PROGRAM MAIN
VAR	
	ipImageMerge		:	ITcVnImage;
	ipImageRed			:	ITcVnImage;
	ipImageBlue			:	ITcVnImage;
	ipImageMergeDisp	:	ITcVnDisplayableImage;
	regionImageDisp	:	ITcVnDisplayableImage;
	
	aBlack				:	TcVnVector4_LREAL := [0, 0, 0];
	aRed				:	TcVnVector4_LREAL := [255, 0, 0];
	aBlue				:	TcVnVector4_LREAL := [0, 0, 255];
	
	aPositionRed		:	TcVnPoint := [20, 20];
	aPositionBlue		:	TcVnPoint := [480, 480];
	bCopyBlue			:	BOOL := FALSE;
	hr: DINT;
END_VAR

//	Disclaimer
  	
//	THIS publication contains statements about the suitability OF our products FOR certain 
//	areas OF application. These statements are based on typical features OF our products. 
//	The examples shown in THIS publication are FOR demonstration purposes only. The 
//	information provided herein should NOT be regarded as specific operation characteristics. 
//	It is incumbent on the customer TO check AND decide whether a product is suitable FOR use 
//	in a particular application. We DO NOT give ANY warranty that the source code which is 
//	made available with this publication is complete or accurate. 
  	
//	THE SAMPLE CODE CONTAINED IN THIS PUBLICATION IS PROVIDED “AS IS” WITHOUT WARRANTY OF ANY 
//	KIND, EITHER EXPRESSED, IMPLIED OR STATUTORY, INCLUDING WITHOUT LIMITATION, ANY WARRANTY 
//	WITH RESPECT TO NON-INFRINGEMENT, FREEDOM FROM PROPRIETARY RIGHTS OF THIRD PARTIES OR 
//	FITNESS FOR ANY PARTICULAR PURPOSE. 
  	
//	THIS publication may be changed FROM TIME TO TIME without prior notice. No liability 
//	is assumed FOR errors AND/OR omissions. Our products are described in detail in our 
//	data sheets AND documentations. Product-specific warnings AND cautions must be observed. 
//	FOR the latest version OF our data sheets AND documentations visit our website 
//	(www.beckhoff.de). 
  	
//	© Beckhoff Automation GmbH & Co. KG, July 2019
  	
//	The reproduction, distribution AND utilization OF THIS document as well as the 
//	communication OF its contents TO others without express authorization is prohibited. 
//	Offenders will be held liable FOR the payment OF damages. All rights reserved in the 
//	event of the grant of a patent, utility model or design.

//	==========================================================================================

//	Sample: Copy Image Region
//	----------------------------------------

// create images & set colors
hr := F_VN_CreateImage(ipImageMerge, 1000, 1000, TCVN_ET_USINT, 3, hr);
hr := F_VN_SetPixels(ipImageMerge, aBlack, hr);
hr := F_VN_CreateImage(ipImageRed, 500, 500, TCVN_ET_USINT, 3, hr);
hr := F_VN_SetPixels(ipImageRed, aRed, hr);
hr := F_VN_CreateImage(ipImageBlue, 500, 500, TCVN_ET_USINT, 3, hr);
hr := F_VN_SetPixels(ipImageBlue, aBlue, hr);

// Copy red image to selected region in merge-image
hr := F_VN_CopyImageRegionToRegion(
	ipSrcImage	:= ipImageRed, 
	nXSrc		:= 0,		nYSrc	:=	0, 
	nWidth		:= 500,		nHeight	:= 500, 
	ipDestImage	:= ipImageMerge, 
	nXDest		:= aPositionRed[0], 
	nYDest		:= aPositionRed[1], 
	hrPrev		:= hr
);

// Copy or mix blue image to selected region in merge-image
hr := F_VN_SetRoi(aPositionBlue[0], aPositionBlue[1], 500, 500, ipImageMerge, hr);
//hr :=F_VN_CopyIntoDisplayableImage(ipImageMerge, regionImageDisp , hr );
hr := F_VN_TransformIntoDisplayableImage(ipImageMerge , regionImageDisp , hr );

IF bCopyBlue THEN
	hr := F_VN_CopyImage(ipImageBlue, ipImageMerge, hr);
ELSE
	hr := F_VN_AddImages(ipImageBlue, ipImageMerge, ipImageMerge, hr);
END_IF
hr := F_VN_ResetRoi(ipImageMerge, hr);

hr := F_VN_CopyIntoDisplayableImage(ipImageMerge, ipImageMergeDisp, hr);

END_PROGRAM

(* stored: Version 1.1.0.1, ProductVersion 3.1.4024.3
   POU MAIN: Id {58583aba-c468-4a32-bbdb-56d33fb53a41}, SpecialFunc None *)
